{attribute addProperty BoxType "KL9260"}
{attribute addProperty Id "Channel_1Channel_0970199100"}
{attribute addProperty CRC "2629167143"}
{attribute addProperty SizeInBites "0"}
{attribute addProperty SizeInBytes "0"}
TYPE KL9260_9CB5E827 :
STRUCT
	{attribute addProperty Name "Channel_1"}
	Channel_1 : Channel_09701991;
END_STRUCT
END_TYPE

(* stored: Version 1.2.0.0, ProductVersion 3.1.4024.9
   DUT KL9260_9CB5E827: Id {e9dcd54e-b90b-45be-8590-c052c0f36f60} *)
